TYPE stParam_ReadQRCode :
STRUCT
	tTimeout		: TIME := T#7S;
END_STRUCT
END_TYPE

(* stored: Version 1.1.0.1, ProductVersion 3.1.4026.18
   DUT stParam_ReadQRCode: Id {ed643308-4ec3-4a60-a022-371297b545be} *)
